{attribute 'Tc2GvlVarNames'}
{attribute 'strict'}
//Stato dell'elemento della lista DI PRODUZIONE
TYPE e_Stato_ElementoLista :
(
	ELEMENTO_NOT_DEFINED 	:= -1, 	//STATO ELEMENTO NON DEFINITO
	ELEMENTO_DA_ELABORARE   := 0,	//STATO ELEMENTO DA ELABORARE
	ELEMENTO_ELABORATO 		:= 1 	//STATO ELEMENTO ELABORATO	
);
END_TYPE
//  ELEMENTO_NOT_DEFINED = '-1'

(* stored: Version 1.1.0.1, ProductVersion 3.1.4024.11
   EnumerationTextList e_Stato_ElementoLista: Id {c9cc5d19-61f8-4177-a2bc-976befbafd80} *)
